TYPE ST_BigBagCmd :
STRUCT
    rBagActualMassManualSet  : REAL;  // wartość wpisana przez operatora
    bApplyBagActualMass      : BOOL;  // przycisk zatwierdzenia (monostabilny)
    bConfirmBagChange        : BOOL;  // potwierdzenie wymiany worka
END_STRUCT
END_TYPE

(* stored: Version 1.1.0.1, ProductVersion 3.1.4024.16
   DUT ST_BigBagCmd: Id {18b4d388-5f80-4074-aeb0-ac9c1e14ee64} *)
